// Implements every optional hook, so all three must resolve non-null.
FUNCTION_BLOCK FakeTestWithAllHooks IMPLEMENTS I_Test, I_TestSetup, I_TestTeardown, I_TestLocation
VAR
	_RunCount : UDINT;
END_VAR

PROPERTY Path : T_MaxString
GET
Path := 'Verifier.Doubles.AllHooks';
END_GET
END_PROPERTY

METHOD Run : BOOL
VAR_INPUT
	Enable : BOOL;
	Test   : I_TestAssertions;
END_VAR
_RunCount := _RunCount + 1;
Run		  := TRUE;
END_METHOD

METHOD Setup : BOOL
VAR_INPUT
	Enable : BOOL;
	Test   : I_TestAssertions;
END_VAR
Setup := TRUE;
END_METHOD

METHOD Teardown : BOOL
VAR_INPUT
	Enable : BOOL;
	Test   : I_TestAssertions;
END_VAR
Teardown := TRUE;
END_METHOD

END_FUNCTION_BLOCK

(* stored: Version 1.1.0.1, ProductVersion 3.1.4026.18
   POU FakeTestWithAllHooks: Id {9eaf8400-c6d8-4d30-9476-6c249e22ec03}, SpecialFunc None
   Folder I_Test: Id {0559658c-8045-46da-9cbd-656683aa0633}
   Folder I_TestLocation: Id {8ae7578a-ca6c-48b6-bb84-13afa4d4eb85}
   Folder I_TestSetup: Id {e096788d-015b-4823-99f2-7d92a9f263b1}
   Folder I_TestTeardown: Id {873a8ee4-3f9c-4116-bd2d-e1850733eb3d}
   Property Path: Id {01241230-534e-4955-aa50-c47993a36a4a}
   Get Get: Id {fbbbda37-212c-43e6-9e19-17b8afd0a931}
   Method Run: Id {9952b636-ad61-4469-b38d-9bdc52cc096c}
   Method Setup: Id {685b444d-fea2-48f8-b0b8-01ea183513b8}
   Method Teardown: Id {a4f86f03-951b-416d-9195-0567dea2f559} *)
